Universal Robots URScript: a_full_bow.script

def a_full_bow():
  global _hidden_verificationVariable=0
  set_standard_analog_input_domain(0, 1)
  set_standard_analog_input_domain(1, 1)
  set_tool_analog_input_domain(0, 1)
  set_tool_analog_input_domain(1, 1)
  set_analog_outputdomain(0, 0)
  set_analog_outputdomain(1, 0)
  set_input_actions_to_default()
  set_gravity([0.0, 0.0, 9.82])
  set_tcp(p[0.028210348281514253,-0.09610723587300697,-0.09969041498611403,0.0,0.0,0.0])
  set_tool_communication(False, 115200, 0, 1, 1.5, 3.5)
  set_tool_output_mode(0)
  set_tool_digital_output_mode(0, 1)
  set_tool_digital_output_mode(1, 1)
  set_tool_voltage(0)
  set_target_payload(0.260000, [0.050000, -0.008000, 0.024000], [0.000163, 0.000163, 0.000163, 0.000000, 0.000000, 0.000000])
  set_safety_mode_transition_hardness(1)
  global Plane_1=p[0.32571614183608727,0.7933870146316717,0.11820742021636722,-2.208244884171713,-0.24738609815952348,-1.9195085473101943]
  global Plane_2=p[0.3436052139151623,0.7478032414335104,0.10077839665899768,2.768545736097797,0.1284831553507919,1.3672805628273381]
  global Plane_3=p[0.31945151854627996,0.6757990361168175,0.09459088830114093,2.7301760593116526,-0.049483824131046385,1.4252239353300047]
  global Plane_4=p[0.3372257363094211,0.6222230974198586,0.07001667903587716,2.621672423508307,-0.12240385890263918,1.4373011913128484]
  # begin: URCap Installation Node
  #   Source: External Control, 1.0.5, FZI Research Center for Information Technology
  #   Type: External Control
  # end: URCap Installation Node
  step_count_6a2d345b_02ef_4768_8296_b2c7f9c3a3e7 = 0.0
  thread Step_Counter_Thread_dbe66d62_ad84_49e2_9f0a_72e40449a578():
    while (True):
      step_count_6a2d345b_02ef_4768_8296_b2c7f9c3a3e7 = step_count_6a2d345b_02ef_4768_8296_b2c7f9c3a3e7 + 1.0
      sync()
    end
  end
  run Step_Counter_Thread_dbe66d62_ad84_49e2_9f0a_72e40449a578()
  global timer_1=0
  global Waypoint_2_p=p[.374968604898, .359127022696, .303034911964, 1.627458665305, 2.337349329242, -1.114572205166]
  global Waypoint_2_q=[-2.7247493443475914, -1.158338378007028, 1.7724153080119223, -1.5486980058846118, -1.9971692127719525, -2.9342161342950686]
  global Waypoint_1_p=p[.277236601206, .734032359319, .156891527665, 1.738924275492, 2.310428552465, -1.107753563859]
  global Waypoint_1_q=[-2.210412708052746, -0.49084595566760747, 0.9551938502229333, -1.302301742823495, -1.605072055336045, -2.4750900912233345]
  global timer_1_is_counting=False
  thread Timer_Thread():
    while (True):
      if (timer_1_is_counting):
        timer_1 = timer_1 + get_steptime()
      end
      sync()
    end
  end
  run Timer_Thread()
  while (True):
    $ 2 "Robot Program"
    $ 3 "bow_dir≔ False "
    global bow_dir=  False
    $ 4 "note_dur≔3"
    global note_dur=3
    $ 5 "timer_1: Start"
    timer_1_is_counting = True
    $ 6 "If bow_dir"
    if (bow_dir):
      $ 7 "MoveL"
      $ 8 "Waypoint_2" "breakAfter"
      global move_thread_flag_8=0
      thread move_thread_8():
        enter_critical
        move_thread_flag_8 = 1
        movel(Waypoint_2_p, a=1.2, v=0.25)
        move_thread_flag_8 = 2
        exit_critical
      end
      move_thread_flag_8 = 0
      move_thread_han_8 = run move_thread_8()
      while (True):
        if (timer_1 == note_dur):
          kill move_thread_han_8
          stopl(1.2)
          $ 9 "Until (expression)"
          break
        end
        sleep(1.0E-10)
        if (move_thread_flag_8 > 1):
          join move_thread_han_8
          break
        end
        sync()
      end
    else:
      $ 10 "Else" "noBreak"
      $ 11 "MoveL"
      $ 12 "Waypoint_1" "breakAfter"
      global move_thread_flag_12=0
      thread move_thread_12():
        enter_critical
        move_thread_flag_12 = 1
        movel(Waypoint_1_p, a=1.2, v=0.25)
        move_thread_flag_12 = 2
        exit_critical
      end
      move_thread_flag_12 = 0
      move_thread_han_12 = run move_thread_12()
      while (True):
        if (timer_1 == note_dur):
          kill move_thread_han_12
          stopl(1.2)
          $ 13 "Until (expression)"
          break
        end
        sleep(1.0E-10)
        if (move_thread_flag_12 > 1):
          join move_thread_han_12
          break
        end
        sync()
      end
    end
    $ 18 "timer_1: Stop"
    timer_1_is_counting = False
    $ 19 "timer_1: Reset"
    timer_1 = 0
  end
end
